// TIA Portal V17 export
// export: Created 2023-12-22T15:08:08.4105318Z, ExportSetting WithDefaults, DisplayName Totally Integrated Automation Portal, DisplayVersion V17, DisplayName TIA Portal Openness, DisplayVersion V17, DisplayName TIA Portal Version Control Interface, DisplayVersion V17, DisplayName STEP 7 Professional, DisplayVersion V17, DisplayName STEP 7 Safety, DisplayVersion V17, DisplayName WinCC Advanced, DisplayVersion V17
FUNCTION_BLOCK "Converter_LAD"   // FB98, LAD
{ S7_Optimized_Access := 'FALSE' }
VERSION : 0.1
// stored: AutoNumber false, IsIECCheckEnabled false, SetENOAutomatically false, UDAEnableTagReadback false
   VAR_INPUT
      Signal : Real;   // Входной сигнал
   END_VAR
   VAR_OUTPUT
      Result : Real;   // Результат линеаризации
   END_VAR
   VAR DB_SPECIFIC
      Use_Min_In { S7_SetPoint := 'True'} : Bool;   // Отсекать входные значения ниже минимума
      Use_Max_In { S7_SetPoint := 'True'} : Bool;   // Отсекать входные значения выше максимума
      Use_Min_Out { S7_SetPoint := 'True'} : Bool;   // Отсекать результат ниже минимума
      Use_Max_Out { S7_SetPoint := 'True'} : Bool;   // Отсекать результат выше максимума
      IO { S7_SetPoint := 'True'} : Bool;   // Входной/Выходной режим
      Inverse { S7_SetPoint := 'True'} : Bool;   // Инверсия выхода
      Min_In { S7_SetPoint := 'True'} : Real;   // Минимальный входной сигнал
      Min_Out { S7_SetPoint := 'True'} : Real;   // Минимальный выходной сигнал
      Max_In { S7_SetPoint := 'True'} : Real;   // Максимальный входной сигнал
      Max_Out { S7_SetPoint := 'True'} : Real;   // Максимальный выходной сигнал
   END_VAR
   VAR_TEMP
      Range_In : Real;   // Диапазон входного сигнала
      Range_Out : Real;   // Диапазон выходного сигнала
      T_T : Real;   // Соотношение диапазонов
      R_Sig : Real;   // Поправка на отрицательные значения
   END_VAR
BEGIN

REGION Network 1: Проверка нижнего уровня входного сигнала
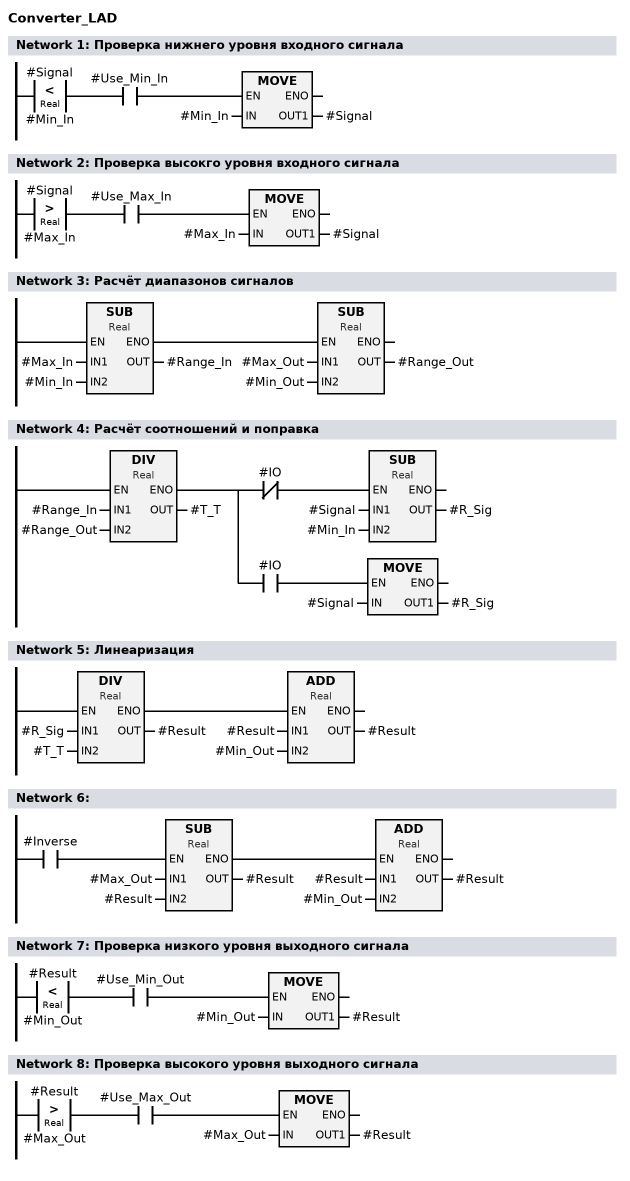
   RUNG wire#powerrail
      { S7_Templates := "SrcType := Real" } LT_Contact(in1 := #Signal, in2 := #Min_In)
      Contact( #Use_Min_In )
      { S7_GenerateENO := "TRUE" } Move(in := #Min_In, out1 => #Signal)
   END_RUNG
   // the same network as SCL:
   IF (#Signal < #Min_In) AND #Use_Min_In THEN #Signal := #Min_In; END_IF;
END_REGION

REGION Network 2: Проверка высокго уровня входного сигнала
   RUNG wire#powerrail
      { S7_Templates := "SrcType := Real" } GT_Contact(in1 := #Signal, in2 := #Max_In)
      Contact( #Use_Max_In )
      { S7_GenerateENO := "TRUE" } Move(in := #Max_In, out1 => #Signal)
   END_RUNG
   // the same network as SCL:
   IF (#Signal > #Max_In) AND #Use_Max_In THEN #Signal := #Max_In; END_IF;
END_REGION

REGION Network 3: Расчёт диапазонов сигналов
   RUNG wire#powerrail
      { S7_Templates := "SrcType := Real"; S7_GenerateENO := "TRUE" } Sub(in1 := #Max_In, in2 := #Min_In, out => #Range_In)
      { S7_Templates := "SrcType := Real"; S7_GenerateENO := "TRUE" } Sub(in1 := #Max_Out, in2 := #Min_Out, out => #Range_Out)
   END_RUNG
   // the same network as SCL:
   // ENO of a box is taken as its EN; it also drops when the box reports an error
   #Range_In := #Max_In - #Min_In;
   #Range_Out := #Max_Out - #Min_Out;
END_REGION

REGION Network 4: Расчёт соотношений и поправка
   RUNG wire#powerrail
      { S7_Templates := "SrcType := Real"; S7_GenerateENO := "TRUE" } Div(in1 := #Range_In, in2 := #Range_Out, out => #T_T)
      wire#w1
      I_Contact( #IO )
      { S7_Templates := "SrcType := Real"; S7_GenerateENO := "TRUE" } Sub(in1 := #Signal, in2 := #Min_In, out => #R_Sig)
   END_RUNG
   RUNG wire#w1
      Contact( #IO )
      { S7_GenerateENO := "TRUE" } Move(in := #Signal, out1 => #R_Sig)
   END_RUNG
   // the same network as SCL:
   // ENO of a box is taken as its EN; it also drops when the box reports an error
   #T_T := #Range_In / #Range_Out;
   IF NOT #IO THEN #R_Sig := #Signal - #Min_In; END_IF;
   IF #IO THEN #R_Sig := #Signal; END_IF;
END_REGION

REGION Network 5: Линеаризация
   RUNG wire#powerrail
      { S7_Templates := "SrcType := Real"; S7_GenerateENO := "TRUE" } Div(in1 := #R_Sig, in2 := #T_T, out => #Result)
      { S7_Templates := "SrcType := Real"; S7_GenerateENO := "TRUE" } Add(in1 := #Result, in2 := #Min_Out, out => #Result)
   END_RUNG
   // the same network as SCL:
   // ENO of a box is taken as its EN; it also drops when the box reports an error
   #Result := #R_Sig / #T_T;
   #Result := #Result + #Min_Out;
END_REGION

REGION Network 6
   RUNG wire#powerrail
      Contact( #Inverse )
      { S7_Templates := "SrcType := Real"; S7_GenerateENO := "TRUE" } Sub(in1 := #Max_Out, in2 := #Result, out => #Result)
      { S7_Templates := "SrcType := Real"; S7_GenerateENO := "TRUE" } Add(in1 := #Result, in2 := #Min_Out, out => #Result)
   END_RUNG
   // the same network as SCL:
   // ENO of a box is taken as its EN; it also drops when the box reports an error
   IF #Inverse THEN
       #Result := #Max_Out - #Result;
       #Result := #Result + #Min_Out;
   END_IF;
END_REGION

REGION Network 7: Проверка низкого уровня выходного сигнала
   RUNG wire#powerrail
      { S7_Templates := "SrcType := Real" } LT_Contact(in1 := #Result, in2 := #Min_Out)
      Contact( #Use_Min_Out )
      { S7_GenerateENO := "TRUE" } Move(in := #Min_Out, out1 => #Result)
   END_RUNG
   // the same network as SCL:
   IF (#Result < #Min_Out) AND #Use_Min_Out THEN #Result := #Min_Out; END_IF;
END_REGION

REGION Network 8: Проверка высокого уровня выходного сигнала
   RUNG wire#powerrail
      { S7_Templates := "SrcType := Real" } GT_Contact(in1 := #Result, in2 := #Max_Out)
      Contact( #Use_Max_Out )
      { S7_GenerateENO := "TRUE" } Move(in := #Max_Out, out1 => #Result)
   END_RUNG
   // the same network as SCL:
   IF (#Result > #Max_Out) AND #Use_Max_Out THEN #Result := #Max_Out; END_IF;
END_REGION
END_FUNCTION_BLOCK
